// TwinCAT 3 PLC project PLC1
// ProgramVersion: 3.1.4024.0
// libraries:
//   Tc2_HVAC, * (Beckhoff Automation GmbH)
//   Tc2_Math, * (Beckhoff Automation GmbH)
//   Tc2_MC2, * (Beckhoff Automation GmbH)
//   Tc2_Standard, * (Beckhoff Automation GmbH)
//   Tc2_System, * (Beckhoff Automation GmbH)
//   Tc2_TcpIp, * (Beckhoff Automation GmbH)
//   Tc2_Utilities, * (Beckhoff Automation GmbH)
//   Tc3_Module, * (Beckhoff Automation GmbH)
// project tree:
//   DUTs/ E_6Axis_Command.TcDUT, E_6Axis_Motion.TcDUT, E_ConnectionSteps.TcDUT, getPosition.TcDUT, Motion_Command_Input.TcDUT, ST_6Axis_State.TcDUT
//   GVLs/ AutoMotionData.TcGVL, GVL.TcGVL
//   / PlcTask.TcTTO
//   POUs/Airbus_TCP/ Deserialize.TcPOU, FB_TCPClient.TcPOU, Serialize.TcPOU
//   POUs/ Buffer.TcPOU, MC_Linear.TcPOU, Kinematics.TcPOU, MAIN.TcPOU, Controller.TcPOU, MathFunc.TcPOU
// real-time tasks:
//   TASK PlcTask: cycle T#2ms, priority 20, ADS port 350
// motion (NC):
//   TASK NC-Task 1 SAF: cycle T#2ms, priority 4, ADS port 501
//   TASK NC-Task 1 SVB: cycle T#10ms, priority 8, ADS port 511
//   AXIS Axis 1 (id 1)
//     Dynamic: AccelerationMaximum=1500, DecelerationMaximum=1500
//     Velo: RefSearch=1, RefSync=1, SlowManual=1, FastManual=3, Maximum=45
//     OtherSettings: AllowMotionCmdToSlave=true
//     encoder EncType=1
//       EncPara: ScaleFactorNumerator=360, ScaleFactorDenominator=104857600, EncMode=3
//         SoftEndMinControl: Enable=true, Range=-180
//         SoftEndMaxControl: Enable=true, Range=180
//     drive DrvType=5
//       Analog: VeloReferenz=50, TorqueSetpointScale=10, ScaleFactorActTorque=0.1
//       TimeComp: TaskDelayCycles=1
//     controller CtrType=1
//       CtrPara: PriorControlFactor=1
//         Observer: BandWidth=20
//   AXIS Axis 2 (id 2)
//     Velo: RefSearch=1, RefSync=1, SlowManual=1, FastManual=3, Maximum=30
//     OtherSettings: AllowMotionCmdToSlave=true
//     encoder EncType=1
//       EncPara: ScaleFactorNumerator=360, ScaleFactorDenominator=104857600, Offset=-0.1609, EncMode=3
//         SoftEndMinControl: Enable=true, Range=-57
//         SoftEndMaxControl: Enable=true, Range=120
//     drive DrvType=5
//       Analog: VeloReferenz=40, TorqueSetpointScale=10, ScaleFactorActTorque=0.1
//       TimeComp: TaskDelayCycles=1
//     controller CtrType=1
//       CtrPara: PriorControlFactor=1
//         Observer: BandWidth=20
//   AXIS Axis 3 (id 3)
//     Velo: RefSearch=1, RefSync=1, SlowManual=1, FastManual=3, Maximum=30
//     OtherSettings: AllowMotionCmdToSlave=true
//     encoder EncType=1
//       EncPara: ScaleFactorNumerator=360, ScaleFactorDenominator=83886080, Offset=2.384, EncMode=3
//         SoftEndMinControl: Enable=true, Range=-125
//         SoftEndMaxControl: Enable=true, Range=55
//     drive DrvType=5
//       Analog: VeloReferenz=40, TorqueSetpointScale=10, ScaleFactorActTorque=0.1
//       TimeComp: TaskDelayCycles=1
//     controller CtrType=1
//       CtrPara: PriorControlFactor=1
//         Observer: BandWidth=20
//   AXIS Axis 4 (id 4)
//     Velo: RefSearch=1, RefSync=1, SlowManual=1, FastManual=3, Maximum=80
//     OtherSettings: AllowMotionCmdToSlave=true
//     encoder EncType=1
//       EncPara: ScaleFactorNumerator=360, ScaleFactorDenominator=83886080, Offset=0.2524, EncMode=3
//         SoftEndMinControl: Enable=true, Range=-180
//         SoftEndMaxControl: Enable=true, Range=180
//     drive DrvType=5
//       Analog: VeloReferenz=100, TorqueSetpointScale=10, ScaleFactorActTorque=0.1
//       TimeComp: TaskDelayCycles=1
//     controller CtrType=1
//       CtrPara: PriorControlFactor=1
//         Observer: BandWidth=20
//   AXIS Axis 5 (id 5)
//     Velo: RefSearch=1, RefSync=1, SlowManual=1, FastManual=3, Maximum=50
//     OtherSettings: AllowMotionCmdToSlave=true
//     encoder EncType=1
//       EncPara: ScaleFactorNumerator=360, ScaleFactorDenominator=64225280, Offset=0.9798, EncMode=3
//         SoftEndMinControl: Enable=true, Range=-95
//         SoftEndMaxControl: Enable=true, Range=95
//     drive DrvType=5
//       Analog: VeloReferenz=60, TorqueSetpointScale=10, ScaleFactorActTorque=0.1
//       TimeComp: TaskDelayCycles=1
//     controller CtrType=1
//       CtrPara: PriorControlFactor=1
//         Observer: BandWidth=20
//   AXIS Axis 6 (id 6)
//     Velo: RefSearch=1, RefSync=1, SlowManual=1, FastManual=3, Maximum=30000
//     OtherSettings: AllowMotionCmdToSlave=true
//     encoder EncType=1
//       EncPara: ScaleFactorNumerator=360, ScaleFactorDenominator=52428800, Offset=-113, EncMode=3
//         SoftEndMinControl: Enable=true, Range=-180
//         SoftEndMaxControl: Enable=true, Range=180
//     drive DrvType=5
//       Analog: VeloReferenz=30000, TorqueSetpointScale=10, ScaleFactorActTorque=0.1
//       TimeComp: TaskDelayCycles=1
//     controller CtrType=1
//       CtrPara: PriorControlFactor=1
//         Observer: BandWidth=20
// I/O:
//   DEVICE Device 2 (EtherCAT) (disabled), AmsNetId 169.254.73.89.3.1
//     Term 1 (R1-EC5500) [R1-EC5500 EtherCAT to E-BUS adapter Module]
//       Term 2 (R1-EC6022) [R1-EC6022 16-ch Sink/Source Type Digital Input Module with 2ms Filter Function]
//       Term 3 (R1-EC7062) [R1-EC7062 16-ch 24VDC/0.5A/Sink Type Digital Output Module]
//       Term 4 (R1-EC8124D0) [R1-EC8124D0 4-ch 16-bit Single-ended/10kHz/Voltage or Current Mode A/D Control Module]
//       Term 11 (EL9011) [EL9011 End Terminal]
//     Drive 5 (SGD7S-xxxxA0x CoE Drive) [SGD7S-xxxxA0x EtherCAT(CoE) SERVOPACK Rev6.01]
//     Drive 6 (SGD7S-xxxxA0x CoE Drive) [SGD7S-xxxxA0x EtherCAT(CoE) SERVOPACK Rev6.01]
//     Drive 7 (SGD7S-xxxxA0x CoE Drive) [SGD7S-xxxxA0x EtherCAT(CoE) SERVOPACK Rev8.19]
//     Drive 8 (SGD7S-xxxxA0x CoE Drive) [SGD7S-xxxxA0x EtherCAT(CoE) SERVOPACK Rev6.01]
//     Drive 9 (SGD7S-xxxxA0x CoE Drive) [SGD7S-xxxxA0x EtherCAT(CoE) SERVOPACK Rev6.01]
//     Drive 10 (SGD7S-xxxxA0x CoE Drive) [SGD7S-xxxxA0x EtherCAT(CoE) SERVOPACK Rev6.01]
// variable links:
//   PLC1/PLC1 Instance <-> NC-Task 1 SAF/Axes/Axis 1
//     PlcTask Inputs/MAIN.SixAxis.Axis[1].NcToPlc <-> Outputs/ToPlc
//     PlcTask Outputs/MAIN.SixAxis.Axis[1].PlcToNc <-> Inputs/FromPlc
//   PLC1/PLC1 Instance <-> NC-Task 1 SAF/Axes/Axis 2
//     PlcTask Inputs/MAIN.SixAxis.Axis[2].NcToPlc <-> Outputs/ToPlc
//     PlcTask Outputs/MAIN.SixAxis.Axis[2].PlcToNc <-> Inputs/FromPlc
//   PLC1/PLC1 Instance <-> NC-Task 1 SAF/Axes/Axis 3
//     PlcTask Inputs/MAIN.SixAxis.Axis[3].NcToPlc <-> Outputs/ToPlc
//     PlcTask Outputs/MAIN.SixAxis.Axis[3].PlcToNc <-> Inputs/FromPlc
//   PLC1/PLC1 Instance <-> NC-Task 1 SAF/Axes/Axis 4
//     PlcTask Inputs/MAIN.SixAxis.Axis[4].NcToPlc <-> Outputs/ToPlc
//     PlcTask Outputs/MAIN.SixAxis.Axis[4].PlcToNc <-> Inputs/FromPlc
//   PLC1/PLC1 Instance <-> NC-Task 1 SAF/Axes/Axis 5
//     PlcTask Inputs/MAIN.SixAxis.Axis[5].NcToPlc <-> Outputs/ToPlc
//     PlcTask Outputs/MAIN.SixAxis.Axis[5].PlcToNc <-> Inputs/FromPlc
//   PLC1/PLC1 Instance <-> NC-Task 1 SAF/Axes/Axis 6
//     PlcTask Inputs/MAIN.SixAxis.Axis[6].NcToPlc <-> Outputs/ToPlc
//     PlcTask Outputs/MAIN.SixAxis.Axis[6].PlcToNc <-> Inputs/FromPlc

CONFIGURATION PLC1
    RESOURCE PLC ON TwinCAT3
        TASK PlcTask(INTERVAL := T#2ms, PRIORITY := 20);
        PROGRAM MAIN WITH PlcTask : MAIN;
    END_RESOURCE
END_CONFIGURATION

// ---- DUTs/E_6Axis_Command.TcDUT
{attribute 'qualified_only'}
{attribute 'strict'}
TYPE E_6Axis_Command :
(
	NO_COMMAND,
	POWER_ON,
	STOP,
	HALT,
	RESET,
	HOMING,
	// Command For Testing
	M_PTP,
	M_DIRE_X,
	M_DIRE_Y,
	M_DIRE_XY,
	M_DIRE_Z,
	M_LINEAR,
	M_CURVE,
	CONSTRUCT, //To build Jenga
	LOOKING,   //To observe Jenga
	TOUCHING,  //To detech Jenga status
	TAKING     //To clamping Jenga
) := NO_COMMAND;
END_TYPE

// ---- DUTs/E_6Axis_Motion.TcDUT
TYPE E_6Axis_Motion :
(
	PTP,
	LINEAR,
	CURVE
);
END_TYPE

// ---- DUTs/E_ConnectionSteps.TcDUT
TYPE E_ConnectionSteps :
(
	eCONNECTION_STATE_IDLE,
	eCONNECTION_STATE_CONNECT_START,
	eCONNECTION_STATE_CONNECT_WAIT,
	eCONNECTION_STATE_DATAEXCHANGE,
	eCONNECTION_STATE_CLOSE_START,
	eCONNECTION_STATE_CLOSE_WAIT,
	eCONNECTION_STATE_ERROR
);
END_TYPE

// ---- DUTs/getPosition.TcDUT
TYPE getPosition :
STRUCT
	a : BYTE;
	b : DINT;
	c : ARRAY[1..6] OF LREAL;
END_STRUCT
END_TYPE

// ---- DUTs/Motion_Command_Input.TcDUT
TYPE Motion_Command_Input :
STRUCT
	mode : E_6Axis_Motion;
	precise : BOOL; // 專門給Homing指令使用
	StartPOS : ARRAY [1..6] OF LREAL;
	FinalPOS : ARRAY [1..6] OF LREAL;
	
END_STRUCT
END_TYPE

// ---- DUTs/ST_6Axis_State.TcDUT
TYPE ST_6Axis_State :
STRUCT
	ready : BOOL;
	busy : BOOL;
	error : BOOL;
	powerOn : BOOL;
	stop : BOOL;
	moving : BOOL;
END_STRUCT
END_TYPE

// ---- GVLs/AutoMotionData.TcGVL
{attribute 'qualified_only'}
VAR_GLOBAL
	POStore : ARRAY [1..2] OF ARRAY [0..100] OF ARRAY [1..6] OF LREAL := [
		[[559, 13, 400, 0, 90, -45]],
		[[561, -43, 400, 0, 90, -135]]];
	MovableBlocks : ARRAY [1..100] OF ARRAY [1..6] OF LREAL; 
	
	CAMStore : ARRAY [1..3] OF ARRAY [0..100] OF ARRAY [1..6] OF LREAL := [
	    [[559, 13, 400, 0, 135, -45]],
		[[561, -43, 400, 0, 135, -135]]]; //姿態要改 
	Heightstore : ARRAY [1..1] OF LREAL ;
END_VAR

// ---- GVLs/GVL.TcGVL
VAR_GLOBAL
	// Software
	isHalt : BOOL;
	InitalPOS : ARRAY [1..6] OF LREAL;

	//Hardward
	input_ana AT %I* : ARRAY[1..8] OF INT;
	output_dig AT %Q* : ARRAY[1..16] OF BOOL;
	input_dig AT %I* : ARRAY[1..16] OF BOOL;
	
	// Extend DATA feat. ADS
	ExtData AT %I* : DINT;
	
	// Extend DATA feat. TCP
	aaa : STRING;
	
END_VAR	
	
VAR_GLOBAL CONSTANT
	// Axes Number
	AXIS_MIN_IDX : USINT := 1;
	AXIS_MAX_IDX : USINT := 6;

	// ADS Setting
	
	// TCP Setting
	PLCPRJ_BUFFER_SIZE						: UDINT := 1000;
	PLCPRJ_SEND_CYCLE_TIME					: TIME := T#1S;
	PLCPRJ_RECEIVE_POLLING_TIME		 		: TIME := T#100MS;
	PLCPRJ_RECEIVE_TIMEOUT					: TIME := T#50S;
	(* Some project specific error codes *)
	PLCPRJ_ERROR_RECEIVE_TIMEOUT			: UDINT := 16#8101;(* Receive timeout error *)
	PLCPRJ_ERROR_SENDFIFO_OVERFLOW			: UDINT := 16#8102;(* Send fifo overflow *)
	PLCPRJ_ERROR_RECFIFO_OVERFLOW			: UDINT := 16#8103;(* Receive fifo overflow *)

END_VAR

// ---- POUs/MAIN.TcPOU
PROGRAM MAIN  
// vision 4.4 *+: TCP, 斜直線移動

VAR
	SixAxis : Controller;
	readA : REAL;
	
	bInit: BOOL := TRUE;
	fbSocketCloseAll: FB_SocketCloseAll; 
	serialize : Serialize;
	deserialize : Deserialize;
	bSocketCloseError: BOOL;
	nSocketCloseError: UDINT;
	
	TCP_Client1     				: FB_TCPClient;
		sClient1SendData			: ARRAY[0..1023] OF BYTE;
		sServer1Host				: T_IPv4Addr;
		nServer1Port				: UDINT;
		bStartClient1Communication	: BOOL 			    := TRUE;
		tClient1CycleTime			: TIME 				:= T#0.5S;
		bClient1SendTrigger			: BOOL;
		bClient1Connected			: BOOL;
		sClient1ReceivedData		: ARRAY[0..1023] OF BYTE;
		bClient1Busy				: BOOL;
		bClientError1				: BOOL;
		nClient1ErrorID1			: UDINT;
		// 新增內容
		rx                          : BYTE;
		mode                        : DINT;
		position                    : ARRAY[1..6] OF LREAL;  // xyzrpy
		tx                          : BYTE;
		fullTime                    : LREAL;
		coeffCopy                   : ARRAY[1..6, 1..6] OF LREAL;
	bAutogenerateData				: BOOL 				:= TRUE;
	fbTimer1						: TON;
	simTime                         : DINT;
	simCoeff                        : ARRAY[1..6] OF LREAL;
	nCnt							: UDINT;	
	
END_VAR

















//	L1 : ARRAY [1..6,1..6] OF LREAL;
//	L2 : ARRAY [1..6,1..6] OF LREAL;
//	L6 : ARRAY [1..6,1..6] OF LREAL;
//	L3,L5 : ARRAY [1..2] OF LREAL;
//	L4 : ARRAY [1..2] OF LREAL := [1, 2];
	
//	i: INT;
//	j: INT;
//	k : Lreal;

SixAxis();
//readA := (INT_TO_REAL(GVL.input_ana[1]) / 32767) * 10;

// Transmission Program
(* On PLC reset or program download close all created/opened sockets/connections *)
// Init Step to close all sockets after login PLC with  downlaod
sServer1Host := '192.168.1.47';
nServer1Port := 200;

IF bInit THEN 			
	fbSocketCloseAll(
		sSrvNetId:= '', 
		bExecute:= TRUE, 
		tTimeout:= T#3S, 
		bBusy=> , 
		bError=> bSocketCloseError, 
		nErrId=> nSocketCloseError);
	IF NOT (fbSocketCloseAll.bBusy OR fbSocketCloseAll.bError) THEN
		bInit := FALSE;
		fbSocketCloseAll(bExecute:= FALSE);
	END_IF
ELSE
	TCP_Client1(
		nRemotePort:= nServer1Port, 								// Server port
		sRemoteHost:= sServer1Host, 								// Server IP (empty for local communication)
		bStartCommunication:= bStartClient1Communication, 			// Start communication, when FALSE, connection is closed
		sSendData:= sClient1SendData, 								// Data that are sent to the server
		tCycleTimeSend:= (*tClient1CycleTime*), 					// TimeInterval for cyclic sending
		bSendTrigger:= ,											// Trigger to send one telegramm manually 
		bConnected => bClient1Connected,							// Switches to TRUE when Client is connected to a server
		sReceivedData=> sClient1ReceivedData,						// Data that are received
		bBusy=> bClient1Busy, 
		bError=> bClientError1, 
		nErrorID=> nClient1ErrorID1, ); 
	deserialize(
		Recvbuffer := sClient1ReceivedData,
		a => rx,
		b => mode,
		c => position);
	
	IF bAutogenerateData AND bClient1Connected THEN
		fbTimer1(IN:= NOT fbTimer1.Q, PT:= tClient1CycleTime, Q=> , ET=> );
		IF fbTimer1.Q  THEN
			IF rx = 84 THEN
				SixAxis.SetMotion(
					mode, SixAxis.HomePoint, position, TRUE, FALSE,
					runTime => fullTime,
					coeffCopy => coeffCopy);
				tx := 67;
				serialize(
					a := tx,
					b := fullTime,
					c := coeffCopy,
					sendbuffer => sClient1SendData);
			
			END_IF
			TCP_Client1.bSendTrigger := TRUE;
			nCnt := nCnt + 1;
		ELSE
			TCP_Client1.bSendTrigger := FALSE;
		END_IF
	END_IF 
END_IF
























// 測試KM
//k := 1.235415445;
//k := LREAL_TO_DINT(k*EXPT(10,2) )/EXPT(10,2);
//FOR i := 1 TO 6 DO
//	FOR j := 1 TO 6 DO
//		IF i <= j THEN
//			L1[i, j] := j;
//		ELSE
//			L1[i, j] := i;
//		END_IF
//	END_FOR
//END_FOR

//FOR i := 1 TO 6 DO
//	FOR j := 1 TO 6 DO
//		IF i <= j THEN
//			L2[i, j] := i*j;
//		ELSE
//			L2[i, j] := i*i;
//		END_IF
//	END_FOR
//END_FOR

////MF.GaussianElimination(base_mat := L1, extend_mat := L2, temp_mat := L6, 6);

END_PROGRAM

// ---- POUs/Controller.TcPOU
FUNCTION_BLOCK Controller

VAR_OUTPUT
	
END_VAR

VAR	
	// 輸入指令，顯示狀態、位置、角度
	command : E_6Axis_Command;	
	state : ST_6Axis_State;
	constructState : UINT;
	touchingState : UINT;
	takeState : UINT;
	JointDegNow : ARRAY [AXIS_MIN_IDX..AXIS_MAX_IDX] OF LREAL;
	PositionNow : ARRAY [AXIS_MIN_IDX..AXIS_MAX_IDX] OF LREAL;
	hasFromCAM : BOOL;
	//StartPosition_Now : ARRAY [AXIS_MIN_IDX..AXIS_MAX_IDX] OF LREAL; // for linear move used
	
	// 開發者使用
	HomePoint : ARRAY [AXIS_MIN_IDX..AXIS_MAX_IDX] OF LREAL := [565, 0, 834, 0, 0, 0];
	HomeJoint : ARRAY [AXIS_MIN_IDX..AXIS_MAX_IDX] OF LREAL := [0, 0, 0, 0, 0, 0]; // for joints space	

	//BufferMot : Motion_Command_Input; // 
	InitalPOS : ARRAY [AXIS_MIN_IDX..AXIS_MAX_IDX] OF LREAL := InitalPOS;
	ActExecute : BOOL := FALSE;
	ExecutePMD : BOOL := FALSE;
	ExecuteCAL : BOOL := FALSE; // 執行一次性計算
 	DIR : LREAL := 0; // XYZ_Direcation XYZ軸方向 = {1:x, 2:y, 3:z, 4:xy, 5:-(xy)}
	PMD : LREAL := 0; // Path_Motion_Displace 路徑移動距離
	TouchDetection : BOOL;
	ZeroArray : ARRAY [AXIS_MIN_IDX..AXIS_MAX_IDX] OF LREAL := [0, 0, 0, 0, 0, 0]; 
	TargetPOS : ARRAY [AXIS_MIN_IDX..AXIS_MAX_IDX] OF LREAL := [650, -150, 500, -42, 0, 45];
	POS_STORAGE : Buffer;

	// 索引
	idx : USINT(AXIS_MIN_IDX..AXIS_MAX_IDX);
	movableBlock_idx : INT;
	i, j : USINT(AXIS_MIN_IDX..AXIS_MAX_IDX);
	z : INT;
	n : ARRAY [1..6] OF LREAL := AutoMotionData.CAMStore[1][0] ;
	usingMotion : INT;
	row, col : INT;
	//ok
	//p : ARRAY [1..2] OF LREAL := AutoMotionData.CAMStore;
	//L : ARRAY [AXIS_MIN_IDX..AXIS_MAX_IDX] OF LREAL ;
	h : INT;
	

	// 基本需要的函式
	Axis : ARRAY[AXIS_MIN_IDX..AXIS_MAX_IDX] OF AXIS_REF;
	Power : ARRAY [AXIS_MIN_IDX..AXIS_MAX_IDX] OF MC_Power;
	Stop : ARRAY [AXIS_MIN_IDX..AXIS_MAX_IDX] OF MC_Stop; //delete
	Halt : ARRAY [AXIS_MIN_IDX..AXIS_MAX_IDX] OF MC_Halt; 
	Reset : ARRAY [AXIS_MIN_IDX..AXIS_MAX_IDX] OF MC_Reset;
	
	// 自訂義函式
	KM : Kinematics;
	MF : MathFunc;
	
	// 移動用函式
	AbsMove : ARRAY [AXIS_MIN_IDX..AXIS_MAX_IDX] OF MC_MoveAbsolute;
	ExtSwitchEn : ARRAY [AXIS_MIN_IDX..AXIS_MAX_IDX] OF MC_ExtSetPointGenEnable;
	ExtSwitchDis : ARRAY [AXIS_MIN_IDX..AXIS_MAX_IDX] OF MC_ExtSetPointGenDisable;
	LinearMove : MC_Linear; 

	// For Curve                         A1  A2  A3  A4  A5  A6
	StartVEL : ARRAY [1..6] OF LREAL := [  0,  0,  0,  0,  0,  0];
	StartACC : ARRAY [1..6] OF LREAL := [  0,  0,  0,  0,  0,  0];
	FinalVEL : ARRAY [1..6] OF LREAL := [  0,  0,  0,  0,  0,  0];
	FinalACC : ARRAY [1..6] OF LREAL := [  0,  0,  0,  0,  0,  0];

	E_Command: INT;
	No_Command: INT;
	PT: TIME;
END_VAR

readAxis();
SetStartPosition();

CASE command OF
	E_6Axis_Command.NO_COMMAND:
		FOR idx := AXIS_MIN_IDX TO AXIS_MAX_IDX DO
			AbsMove[idx].Execute := FALSE;
		END_FOR
		isHalt := FALSE;
		ExecutePMD := FALSE;
		constructState := 0;
		ActExecute := FALSE;
		
	E_6Axis_Command.POWER_ON:
		FOR idx := AXIS_MIN_IDX TO AXIS_MAX_IDX DO
			Power[idx].Enable := TRUE;
		END_FOR
		IF state.powerOn THEN
			command := E_6Axis_Command.HOMING;
		END_IF
	
	E_6Axis_Command.HALT:
		FOR idx := AXIS_MIN_IDX TO AXIS_MAX_IDX DO
			Halt[idx].Execute := TRUE;
		END_FOR
		IF NOT state.moving THEN
			FOR idx := AXIS_MIN_IDX TO AXIS_MAX_IDX DO
				Halt[idx].Execute := FALSE;
			END_FOR
		END_IF
		command := E_6axis_Command.NO_COMMAND;
	
	E_6Axis_Command.RESET:
		FOR idx := AXIS_MIN_IDX TO AXIS_MAX_IDX DO
			Reset[idx].Execute := TRUE;
			IF Reset[idx].Done THEN
				Reset[idx].Execute := FALSE;
			END_IF
		END_FOR
		command := E_6axis_Command.NO_COMMAND;

	// SetMotion(路徑模式，起點，終點，FALSE);		
	E_6Axis_Command.HOMING:
		ActExecute := TRUE;
		SetMotion(0, InitalPOS, HomeJoint, FALSE, TRUE);
		IF NOT ActExecute THEN
			command := E_6axis_Command.NO_COMMAND;
		END_IF

	E_6Axis_Command.M_PTP:
		ActExecute := TRUE;
		SetMotion(0, InitalPOS, TargetPOS, FALSE, FALSE);
		IF NOT ActExecute THEN
			command := E_6axis_Command.NO_COMMAND;
		END_IF
		
	E_6Axis_Command.M_DIRE_X:
		IF NOT ExecutePMD THEN
			MF.VectorMotionPOS(POS := TargetPOS, DIR, PMD);
			ExecutePMD := TRUE;
		END_IF
		ActExecute := TRUE;
		SetMotion(1, InitalPOS, TargetPOS, FALSE, FALSE);
		IF NOT ActExecute THEN
			command := E_6axis_Command.NO_COMMAND;
		END_IF
		
	E_6Axis_Command.M_DIRE_Y:
		IF NOT ExecutePMD THEN
			MF.VectorMotionPOS(POS := TargetPOS, DIR, PMD);
			ExecutePMD := TRUE;
		END_IF
		ActExecute := TRUE;
		SetMotion(1, InitalPOS, TargetPOS, FALSE, FALSE);
		IF NOT ActExecute THEN
			command := E_6axis_Command.NO_COMMAND;
		END_IF
	
	E_6Axis_Command.M_DIRE_XY:
		IF NOT ExecutePMD THEN
			MF.VectorMotionPOS(POS := TargetPOS, DIR, PMD);
			ExecutePMD := TRUE;
		END_IF
		ActExecute := TRUE;
		SetMotion(1, InitalPOS, TargetPOS, FALSE, FALSE);
		IF NOT ActExecute THEN
			command := E_6axis_Command.NO_COMMAND;
		END_IF
		
	E_6Axis_Command.M_DIRE_Z:
		IF NOT ExecutePMD THEN
			MF.VectorMotionPOS(POS := TargetPOS, DIR, PMD);
			ExecutePMD := TRUE;
		END_IF
		ActExecute := TRUE;
		SetMotion(1, InitalPOS, TargetPOS, FALSE, FALSE);
		IF NOT ActExecute THEN
			command := E_6axis_Command.NO_COMMAND;
		END_IF
		
	E_6Axis_Command.M_LINEAR:
		ActExecute := TRUE;
		SetMotion(1, InitalPOS, TargetPOS, FALSE, FALSE);
		IF NOT ActExecute THEN
			command := E_6axis_Command.NO_COMMAND;
		END_IF
		
	E_6Axis_Command.M_CURVE:
		ActExecute := TRUE;
		SetMotion(2, InitalPOS, TargetPOS, FALSE, FALSE);
		IF NOT ActExecute THEN
			command := E_6axis_Command.NO_COMMAND;
		END_IF
		
	E_6Axis_Command.TOUCHING://判斷式
		IF NOT ActExecute THEN
			CASE touchingState OF
				0: //要再加一個判斷式判斷是哪一個位置
					//z := z + 1;            // 疊疊樂右面與左面
					usingMotion := 2;
					
					IF z = 1 THEN
						TargetPOS[1]:= n[1];
						TargetPOS[2]:= n[2];
						TargetPOS[3]:= 500;
						TargetPOS[4]:= 0;
						TargetPOS[5]:= 90;
						TargetPOS[6]:= -45;
					ELSIF z = 2 THEN
						TargetPOS[1]:= n[1];
						TargetPOS[2]:= n[2];
						TargetPOS[3]:= 500;
						TargetPOS[4]:= 0;
						TargetPOS[5]:= 90;
						TargetPOS[6]:= -135;
					END_IF
					      // 移動模式
					//TargetPOS := AutoMotionData.CAMStore[n][z];  // n=0
					//n := n + 1;
					touchingState := touchingState + 1;
				1:
					usingMotion := 1;
					IF z = 1 THEN
						MF.VectorMotionPOS(POS := TargetPOS, 5, -25);
					ELSIF z = 2 THEN
						MF.VectorMotionPOS(POS := TargetPOS, 4, 25);
					END_IF
					//AutoMotionData.POStore[z][n] := TargetPOS;
					//n := n + 1;
					touchingState := touchingState + 1;
				2: 
					usingMotion := 1;
					IF z = 1 THEN
						MF.VectorMotionPOS(POS := TargetPOS, 3, -(500-n[3]));
					ELSIF z = 2 THEN
						MF.VectorMotionPOS(POS := TargetPOS, 3, -(500-n[3]));
					END_IF
					touchingState := touchingState + 1;
				3:
					PT := T#1S;
					input_dig[1] := TRUE;
					PT := T#1S;
					//加計時器
					input_dig[1] := FALSE;
				4:
					usingMotion := 1;
					IF z = 1 THEN
						MF.VectorMotionPOS(POS := TargetPOS, 3, (500-n[3]));
					ELSIF z = 2 THEN
						MF.VectorMotionPOS(POS := TargetPOS, 3, (500-n[3]));
					END_IF
					touchingState := touchingState + 1;
				
				5:
					command := E_6axis_Command.HOMING;
					touchingState := touchingState + 1;
				6:
					command := E_6axis_Command.TAKING;
			END_CASE			
		END_IF
	SetMotion(usingMotion, InitalPOS, TargetPOS, FALSE, FALSE);
	
	E_6Axis_Command.TAKING:
		IF NOT ActExecute THEN
			CASE takeState OF
				0:
					usingMotion := 1;
					input_dig[2] := FALSE;
					
					IF z = 1 THEN
						MF.VectorMotionPOS(POS := TargetPOS, 5, (n[1]+100));
						MF.VectorMotionPOS(POS := TargetPOS, 5, (n[2]+100));
						TargetPOS[3] := 500;
						TargetPOS[4] := 0;
						TargetPOS[5] := -90;
						TargetPOS[6] := 45;
					ELSIF z = 2 THEN
						MF.VectorMotionPOS(POS := TargetPOS, 4, (n[1]-100));
						MF.VectorMotionPOS(POS := TargetPOS, 4, (n[2]-100));
						TargetPOS[3] := 500;
						TargetPOS[4] := 0;
						TargetPOS[5] := -90;
						TargetPOS[6] := -135;
						
					END_IF
					touchingState := touchingState + 1;	
				1:
					usingMotion := 1;
					IF z = 1 THEN
						MF.VectorMotionPOS(POS := TargetPOS, 3, -(500-n[3]));
					ELSIF z = 2 THEN
						MF.VectorMotionPOS(POS := TargetPOS, 3, -(500-n[3]));
					END_IF
					//AutoMotionData.POStore[z][n] := hasFromCAM;
					//n := n + 1;
					touchingState := touchingState + 1;
				2:
					usingMotion := 1; 
					input_dig[2]:= TRUE ;
					PT := T#1S;
					touchingState := touchingState + 1;
				3:
					usingMotion := 1; 
					IF z = 1 THEN
						MF.VectorMotionPOS(POS := TargetPOS, 5, 30);
					ELSIF z = 2 THEN
						MF.VectorMotionPOS(POS := TargetPOS, 4, -30);
					END_IF
					touchingState := touchingState + 1;
				4:
					usingMotion := 1;
					
					MF.VectorMotionPOS(POS := TargetPOS, 3, (AutoMotionData.Heightstore[1]-n[3]+2));
					touchingState := touchingState + 1;
				5:
				   IF z = 1 THEN
						MF.VectorMotionPOS(POS := TargetPOS, 5, -60);
					ELSIF z = 2 THEN
						MF.VectorMotionPOS(POS := TargetPOS, 4, 60);
					END_IF
					PT := T#1S;
					input_dig[2]:= FALSE ;
					touchingState := touchingState + 1;
				6:
					command := E_6axis_Command.HOMING;
					
			END_CASE
		END_IF
		SetMotion(usingMotion, InitalPOS, TargetPOS, FALSE, FALSE);
		ActExecute := TRUE;
				
				
//	E_6Axis_Command.LOOKING:
//		SetMotion(0, InitalPOS, TargetPOS, FALSE);

END_CASE

Decider();
Update_AbsMove_Motion();
Update_Custom_Motion();
ActPower();
ActReset();
ActStop();

//	E_6Axis_Command.CONSTRUCT:
//		IF NOT ActExecute THEN
//			CASE constructState OF
//				0:
//					z := z + 1;            // 疊疊樂右面與左面
//					usingMotion := 2;      // 移動模式
//					TargetPOS := AutoMotionData.POStore[z][n];  // n=0
//					n := n + 1;
//					constructState := constructState + 1;
//				1:
//					usingMotion := 1;
//					IF z = 1 THEN
//						MF.VectorMotionPOS(POS := TargetPOS, 4, 90);
//					ELSIF z = 2 THEN
//						MF.VectorMotionPOS(POS := TargetPOS, 5, 90);
//					END_IF
//					AutoMotionData.POStore[z][n] := TargetPOS;
//					n := n + 1;
//					constructState := constructState + 1;
//				2:
//					usingMotion := 1;
//					IF z = 1 THEN
//						MF.VectorMotionPOS(POS := TargetPOS, 3, -95);
//					ELSIF z = 2 THEN
//						MF.VectorMotionPOS(POS := TargetPOS, 3, -110);
//					END_IF					
//					AutoMotionData.POStore[z][n] := TargetPOS;
//					n := n + 1;
//					constructState := constructState + 1;
//				3:
//					usingMotion := 1;
//					TouchDetection := TRUE;
//					ExecuteCAL := FALSE;
//					IF z = 1 THEN
//						MF.VectorMotionPOS(POS := TargetPOS, 4, -40);
//					ELSIF z = 2 THEN
//						MF.VectorMotionPOS(POS := TargetPOS, 5, -40);
//					END_IF	
//					AutoMotionData.POStore[z][n] := TargetPOS;
//					n := n + 1;
//					movableBlock_idx := movableBlock_idx + 1;
//					constructState := constructState + 1;
//				4:
//					usingMotion := 1;
//					TouchDetection := FALSE;
//					row := row + 1;
//					IF z = 1 THEN
//						MF.VectorMotionPOS(POS := TargetPOS, 4, 40);
//					ELSIF z = 2 THEN
//						MF.VectorMotionPOS(POS := TargetPOS, 5, 40);
//					END_IF	
//					AutoMotionData.POStore[z][n] := TargetPOS;
//					n := n + 1; 
//					constructState := constructState + 1;
//					IF row = 3 THEN
//						row := 0;
//						constructState := 6;
//						col := col + 1;
//						IF col = 4 THEN
//							constructState := 8;
//						END_IF
//					END_IF
//				5:
//					usingMotion := 1;
//					IF z = 1 THEN
//						MF.VectorMotionPOS(POS := TargetPOS, 5, -25);
//					ELSIF z = 2 THEN
//						MF.VectorMotionPOS(POS := TargetPOS, 4, -25);
//					END_IF	
//					AutoMotionData.POStore[z][n] := TargetPOS;
//					n := n + 1;
//					constructState := 3;
//				6:
//					usingMotion := 1;
//					MF.VectorMotionPOS(POS := TargetPOS, 3, -30);
//					AutoMotionData.POStore[z][n] := TargetPOS;
//					n := n + 1;
//					constructState := constructState + 1;
//				7:
//					usingMotion := 1;
//					IF z = 1 THEN
//						MF.VectorMotionPOS(POS := TargetPOS, 5, 50);
//					ELSIF z = 2 THEN
//						MF.VectorMotionPOS(POS := TargetPOS, 4, 50);
//					END_IF	
//					AutoMotionData.POStore[z][n] := TargetPOS;
//					n := n + 1;
//					constructState := 3;
//				8:
//					usingMotion := 2;
//					TargetPOS := AutoMotionData.POStore[z][1];
//					constructState := 9;
//				9:
//					usingMotion := 2;
//					TargetPOS := HomePoint;
//					n := 0;
//					row := 0;
//					col := 0;
//					constructState := 0;
//					IF z = 2 THEN
//						constructState := 10;
//					END_IF
//				10:
//					command := E_6axis_Command.HOMING;
//					constructState := 11;
//			END_CASE
//		END_IF
//		ActExecute := TRUE;
//		IF TouchDetection THEN
//			IF input_dig[1] THEN
//				IF NOT ExecuteCAL THEN
//					AutoMotionData.MovableBlocks[movableBlock_idx] := ZeroArray;
//					movableBlock_idx := movableBlock_idx - 1;
//					ExecuteCAL := TRUE;
//				END_IF
//			ELSE
//				// 減2是為了擷取上一個座標
//				AutoMotionData.MovableBlocks[movableBlock_idx] := AutoMotionData.POStore[z][n-2];
//			END_IF
//		END_IF

//		IF NOT (constructState = 11) THEN
//			SetMotion(usingMotion, InitalPOS, TargetPOS, FALSE, FALSE);
//		ELSE
//			z := 0;
//		END_IF

ACTION ActHalt:
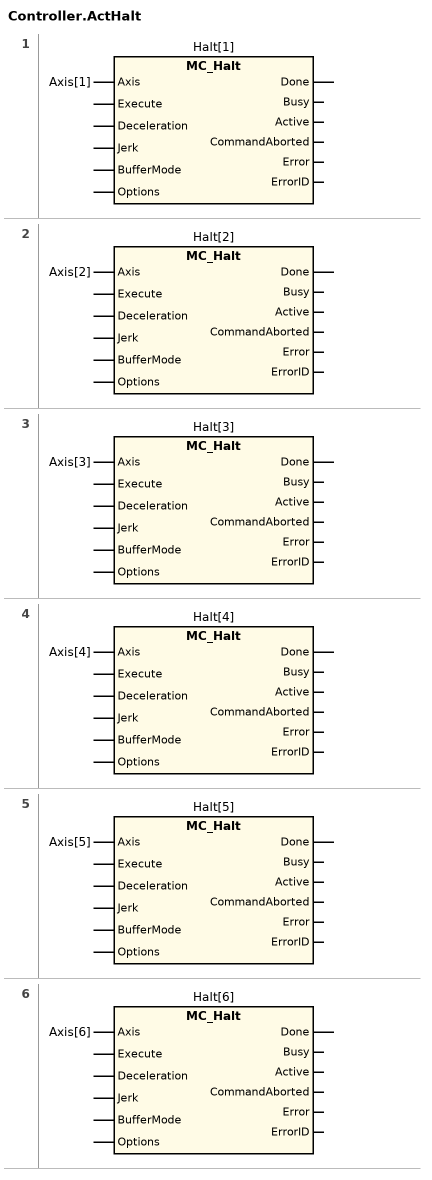
// NETWORK 1
Halt[1](Axis := Axis[1]); // MC_Halt

// NETWORK 2
Halt[2](Axis := Axis[2]); // MC_Halt

// NETWORK 3
Halt[3](Axis := Axis[3]); // MC_Halt

// NETWORK 4
Halt[4](Axis := Axis[4]); // MC_Halt

// NETWORK 5
Halt[5](Axis := Axis[5]); // MC_Halt

// NETWORK 6
Halt[6](Axis := Axis[6]); // MC_Halt
END_ACTION

ACTION ActPower:
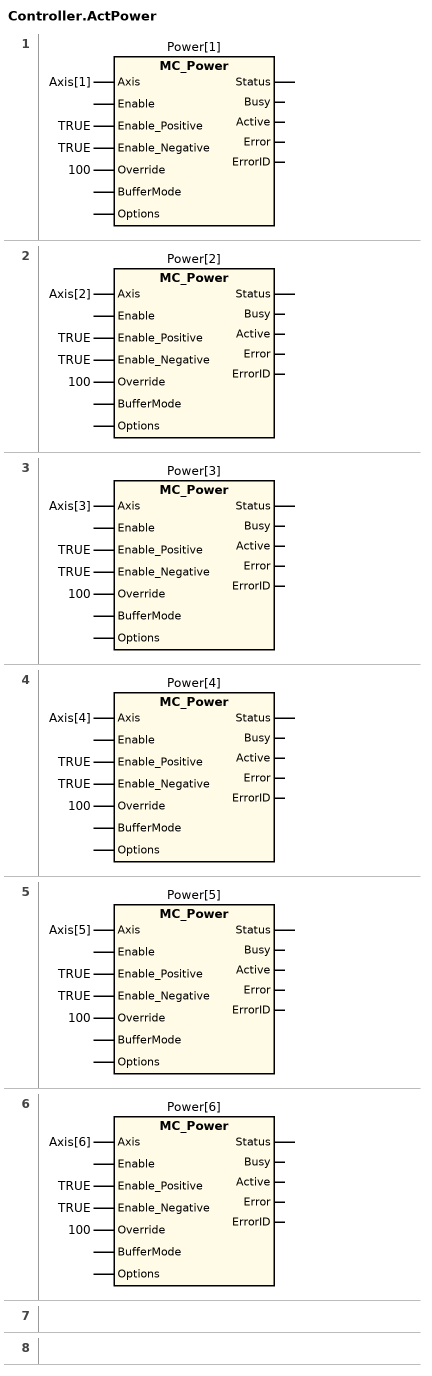
// NETWORK 1
Power[1](Axis := Axis[1], Enable_Positive := TRUE, Enable_Negative := TRUE, Override := 100); // MC_Power

// NETWORK 2
Power[2](Axis := Axis[2], Enable_Positive := TRUE, Enable_Negative := TRUE, Override := 100); // MC_Power

// NETWORK 3
Power[3](Axis := Axis[3], Enable_Positive := TRUE, Enable_Negative := TRUE, Override := 100); // MC_Power

// NETWORK 4
Power[4](Axis := Axis[4], Enable_Positive := TRUE, Enable_Negative := TRUE, Override := 100); // MC_Power

// NETWORK 5
Power[5](Axis := Axis[5], Enable_Positive := TRUE, Enable_Negative := TRUE, Override := 100); // MC_Power

// NETWORK 6
Power[6](Axis := Axis[6], Enable_Positive := TRUE, Enable_Negative := TRUE, Override := 100); // MC_Power

// NETWORK 7

// NETWORK 8
END_ACTION

ACTION ActReset:
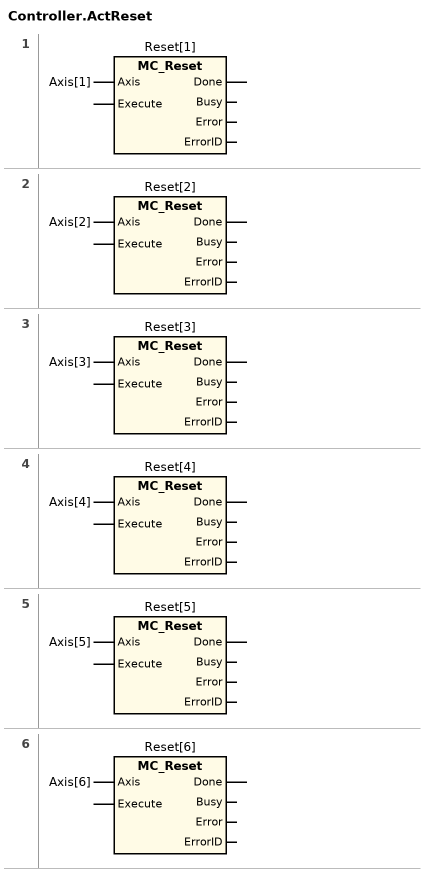
// NETWORK 1
Reset[1](Axis := Axis[1]); // MC_Reset

// NETWORK 2
Reset[2](Axis := Axis[2]); // MC_Reset

// NETWORK 3
Reset[3](Axis := Axis[3]); // MC_Reset

// NETWORK 4
Reset[4](Axis := Axis[4]); // MC_Reset

// NETWORK 5
Reset[5](Axis := Axis[5]); // MC_Reset

// NETWORK 6
Reset[6](Axis := Axis[6]); // MC_Reset
END_ACTION

ACTION ActStop:
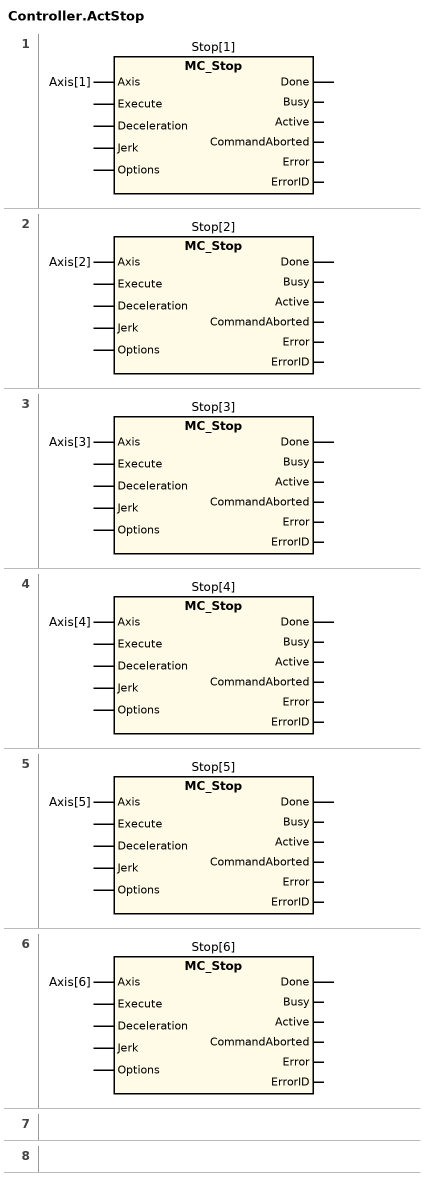
// NETWORK 1
Stop[1](Axis := Axis[1]); // MC_Stop

// NETWORK 2
Stop[2](Axis := Axis[2]); // MC_Stop

// NETWORK 3
Stop[3](Axis := Axis[3]); // MC_Stop

// NETWORK 4
Stop[4](Axis := Axis[4]); // MC_Stop

// NETWORK 5
Stop[5](Axis := Axis[5]); // MC_Stop

// NETWORK 6
Stop[6](Axis := Axis[6]); // MC_Stop

// NETWORK 7

// NETWORK 8
END_ACTION

ACTION Decider:
IF NOT state.moving AND AbsMove[1].Done AND AbsMove[2].Done AND AbsMove[3].Done AND AbsMove[4].Done  AND AbsMove[5].Done AND AbsMove[6].Done THEN
	command := E_6axis_Command.NO_COMMAND;	
END_IF

IF state.error THEN
	command := E_6Axis_Command.RESET;
END_IF

IF isHalt THEN
	command := E_6Axis_Command.HALT;
END_IF
END_ACTION

METHOD mode_Curve : BOOL

VAR_INPUT
	six_mat : ARRAY [1..6, 1..6] OF LREAL;
END_VAR

VAR_OUTPUT
	execute_fullTime : LREAL;
	coeffCopy : ARRAY [1..6, 1..6] OF LREAL;
END_VAR

VAR
	idx : DINT;
	i, j : INT;
	t : LREAL;
	temp : LREAL; // 導正係數用
	
	startAngles : ARRAY [1..6] OF LREAL;
	finalAngles : ARRAY [1..6] OF LREAL;
	pos01, pos02 : ARRAY [1..3] OF LREAL; //start and final point for calculate fulltime
	
	six_matCopy : ARRAY [1..6, 1..6] OF LREAL;
	TimeMatrix : ARRAY [1..6, 1..6] OF LREAL;
END_VAR
// Angles_mat
six_matCopy := six_mat;  // 含有角度 := 含有座標
FOR idx := 1 TO 6 DO 
	IF (idx < 3) THEN
		pos01[idx] := six_mat[idx, 1];
		pos02[idx] := six_mat[idx, 4];
	END_IF
	startAngles[idx] := six_mat[idx, 1];
	finalAngles[idx] := six_mat[idx, 4];
END_FOR
KM.Inverse(position := startAngles, degrees => startAngles);
KM.Inverse(position := finalAngles, degrees => finalAngles);
FOR idx := 1 TO 6 DO 
	six_matCopy[idx, 1] := startAngles[idx];
	six_matCopy[idx, 4] := finalAngles[idx];
END_FOR

MF.FindFullTime(pos01, pos02, 10, execute_fullTime => execute_fullTime);
t := execute_fullTime;
// Time_mat
FOR i := 1 TO 6 DO
    FOR j := 1 TO 6 DO
        CASE j OF
            1: 
                // 第一列固定為1、0、0、0、0、0
                TimeMatrix[i, j] := SEL(i = 1, 0, 1);
            2: 
                // 第二列固定為0、1、0、0、0、0
                TimeMatrix[i, j] := SEL(i = 2, 0, 1);
            3:
                // 第三列固定為0、0、2、0、0、0
                TimeMatrix[i, j] := SEL(i = 3, 0, 2);
            4:
                // 第四列公式：1 * EXPT(t, i)
                TimeMatrix[i, j] := EXPT(t, i-1);
            5:
                // 第五列公式：i * EXPT(t, i-1)
                TimeMatrix[i, j] := (i-1) * EXPT(t, i-2);
            6:
                // 第六列公式：(i * (i - 1)) * EXPT(t, i-2)
                TimeMatrix[i, j] := (i-1) * (i-2) * EXPT(t, i-3);
        END_CASE
    END_FOR
END_FOR

MF.GaussianElimination(base_mat := TimeMatrix, extend_mat := six_matCopy, temp_mat := coeffCopy, 6); //inverse 會搞壞原本的東西

FOR i := 1 TO 6 DO
	FOR j := 1 TO 3 DO
		temp := coeffCopy[i, j];
		coeffCopy[i, j] := coeffCopy[i, 7-j];
		coeffCopy[i, 7-j] := temp;
	END_FOR		
END_FOR
END_METHOD

METHOD mode_Linear : BOOL

VAR_INPUT
	six_pos : ARRAY [1..6, 1..6] OF LREAL;
END_VAR

VAR_OUTPUT
	execute_fullTime : LREAL;
	coeffCopy : ARRAY [1..6, 1..6] OF LREAL;
END_VAR

VAR
	idx : DINT;
	i, j : DINT;
	temp : LREAL; // 導正係數用

	pos01, pos02 : ARRAY [1..3] OF LREAL; //start and final point
	temp_pos : ARRAY [1..6] OF LREAL;
	temp_ang : ARRAY [1..6] OF LREAL;
	six_pos_angles : ARRAY [1..6, 1..6] OF LREAL;
	
	six_time : ARRAY [1..6, 1..6] OF LREAL;
	timeCopy : ARRAY [1..6, 1..6] OF LREAL;
	
END_VAR
// Angles_mat
FOR i := 1 TO 6 DO
	FOR j := 1 TO 6 DO
		temp_pos[j] := six_pos[i, j];
	END_FOR
	KM.Inverse(position := temp_pos, degrees => temp_ang);
	FOR j := 1 TO 6 DO
		six_pos_angles[j, i] := temp_ang[j];
	END_FOR
END_FOR

FOR idx := 1 TO 3 DO 
	pos01[idx] := six_pos[1, idx];
	pos02[idx] := six_pos[6, idx];
END_FOR
MF.FindFullTime(pos01, pos02, 10, execute_fullTime => execute_fullTime);

// Time_mat
FOR i := 1 TO 6 DO
	six_time[1, i] := 1;
	six_time[2, i] := (execute_fullTime)/5 * (i-1);
	FOR j := 3 TO 6 DO
		six_time[j, i] := EXPT(six_time[2, i], j-1);
	END_FOR
END_FOR

FOR i := 1 TO 6 DO
	FOR j := 1 TO 6 DO
		coeffCopy[i, j] := 0; // clear temp
		timeCopy[i, j] := six_time[i, j];
	END_FOR
END_FOR

MF.GaussianElimination(base_mat := timeCopy, extend_mat := six_pos_angles, temp_mat := coeffCopy, 6); //inverse 會搞壞原本的東西

FOR i := 1 TO 6 DO
	FOR j := 1 TO 3 DO
		temp := coeffCopy[i, j];
		coeffCopy[i, j] := coeffCopy[i, 7-j];
		coeffCopy[i, 7-j] := temp;
	END_FOR		
END_FOR
END_METHOD

METHOD mode_PTP : BOOL

VAR_INPUT
	angles01 : ARRAY [1..6] OF LREAL; // start position (degree)
	angles02 : ARRAY [1..6] OF LREAL; // final position (degree)
END_VAR

VAR
	idx : DINT;
	
	longest_distance : LREAL := 0;
	//time_factor : LREAL;
	execute_fullTime : LREAL := 3;
	
END_VAR
//// Execute Time
//FOR idx := 1 TO 6 DO
//	longest_distance := MAX(longest_distance, ABS(angles02[idx] - angles01[idx]));
//END_FOR
//time_factor := EXPT(30, -1); // The larger the denominator, the faster the speed
//execute_fullTime := time_factor * longest_distance;
//execute_fullTime := LREAL_TO_DINT(execute_fullTime * 1000)/1000; // Adjust Time
//IF execute_fullTime < 0.01 THEN
//	execute_fullTime := 3;
//END_IF

FOR idx := 1 TO 6 DO
	AbsMove[idx].Position := angles02[idx];
	AbsMove[idx].Velocity := ABS(angles02[idx] - Axis[idx].NcToPlc.ActPos) / execute_fullTime;
	IF AbsMove[Idx].Velocity < 0.001 THEN
		AbsMove[Idx].Velocity := 0.001;  // Module Minium Limit
	END_IF
END_FOR
END_METHOD

METHOD readAxis : BOOL

VAR
	
END_VAR
FOR idx := AXIS_MIN_IDX TO AXIS_MAX_IDX DO
	Axis[idx]();
	JointDegNow[idx] := Axis[idx].NcToPlc.ActPos;
END_FOR
KM.Forward(angles := JointDegNow, position => PositionNow);

state.powerOn := Power[1].Status AND Power[2].Status AND Power[3].Status AND Power[4].Status AND Power[5].Status AND Power[6].Status;
state.stop := Stop[1].Done AND Stop[2].Done AND Stop[3].Done AND Stop[4].Done AND Stop[5].Done AND Stop[6].Done;
state.moving := Axis[1].Status.Moving OR Axis[2].Status.Moving OR Axis[3].Status.Moving OR  Axis[4].Status.Moving OR Axis[5].Status.Moving OR Axis[6].Status.Moving;
//state.pause := NOT (state.moving OR state.stop);
state.error := Axis[1].Status.Error OR Axis[2].Status.Error OR Axis[3].Status.Error OR Axis[4].Status.Error OR Axis[5].Status.Error OR Axis[6].Status.Error;
END_METHOD

METHOD SetMotion : BOOL

VAR_INPUT
	mode : DINT;
	StartPOS : ARRAY [1..6] OF LREAL;
	FinalPOS : ARRAY [1..6] OF LREAL;
	isSIM : BOOL;
	precise : BOOL; // 專門給Homing指令使用
	
END_VAR

VAR_OUTPUT
	runTime : LREAL;
	coeffCopy : ARRAY[1..6, 1..6] OF LREAL;
END_VAR

VAR
	// PTP
	ptpAngles_01 : ARRAY [1..6] OF LREAL;
	ptpAngles_02 : ARRAY [1..6] OF LREAL;
	
	// Linear
	six_pos : ARRAY [1..6, 1..6] OF LREAL;

	
	// Curve 
	six_mat : ARRAY [1..6, 1..6] OF LREAL;
	
	// Linear & Curve
	customAngles : ARRAY [1..6] OF LREAL;  // deg & rad

	PTPMove_done : BOOL;
END_VAR


CASE mode OF
	0: // PTP
		FOR idx := AXIS_MIN_IDX TO AXIS_MAX_IDX DO
			AbsMove[idx].Execute := TRUE;
			IF NOT precise THEN
				KM.Inverse(position := StartPOS, degrees => ptpAngles_01);
				KM.Inverse(position := FinalPOS, degrees => ptpAngles_02);
				mode_PTP(ptpAngles_01, ptpAngles_02);
			ELSE
				AbsMove[idx].Position := HomeJoint[idx];
				AbsMove[idx].Velocity := 5;
			END_IF
		END_FOR		
		
		PTPMove_done := TRUE;
		FOR idx := 1 TO 6 DO
			IF NOT AbsMove[idx].Done THEN
				PTPMove_done := FALSE;
				EXIT;
			END_IF
		END_FOR
		
	1: // LINEAR
		KM.Inverse(position := FinalPOS, degrees => customAngles);
								
		FOR idx := AXIS_MIN_IDX TO AXIS_MAX_IDX DO
			ExtSwitchEn[idx].Position := customAngles[idx];
			ExtSwitchEn[idx].Execute := TRUE;
			ExtSwitchDis[idx].Execute := FALSE;
		END_FOR
		
		MF.FindForSixPoints(StartPOS, FinalPOS, six_pos => six_pos);
		mode_Linear(six_pos, coeffCopy => coeffCopy, execute_fullTime => runTime);
		
		LinearMove.Execute := TRUE;
		LinearMove.CoeffCopy := coeffCopy;
		LinearMove.RunTime := runTime;
	
	2: // CURVE
		KM.Inverse(position := FinalPOS, degrees => customAngles);
		
		FOR idx := AXIS_MIN_IDX TO AXIS_MAX_IDX DO
			ExtSwitchEn[idx].Position := customAngles[idx];
			ExtSwitchEn[idx].Execute := TRUE;
			ExtSwitchDis[idx].Execute := FALSE;
		END_FOR

		FOR idx := AXIS_MIN_IDX TO AXIS_MAX_IDX DO
			six_mat[idx, 1] :=  StartPOS[idx];
			six_mat[idx, 2] :=  StartVEL[idx];
			six_mat[idx, 3] :=  StartACC[idx];
			six_mat[idx, 4] :=  FinalPOS[idx];
			six_mat[idx, 5] :=  FinalVEL[idx];
			six_mat[idx, 6] :=  FinalACC[idx];
		END_FOR
		mode_Curve(six_mat, coeffCopy => coeffCopy, execute_fullTime => runTime);
		
		LinearMove.Execute := TRUE;
		LinearMove.CoeffCopy := coeffCopy;
		LinearMove.RunTime := runTime;
END_CASE

IF NOT isSIM AND (PTPMove_done OR LinearMove.Done) THEN
	// SetStartPosition
	IF precise THEN
		InitalPOS := HomePoint;
	ELSE

		LinearMove.Execute := FALSE;
		//running := FALSE;
		FOR idx := AXIS_MIN_IDX TO AXIS_MAX_IDX DO
			AbsMove[idx].Execute := FALSE;
			ExtSwitchEn[idx].Execute := FALSE;
			ExtSwitchDis[idx].Execute := TRUE;
		END_FOR
		InitalPOS := FinalPOS;
	END_IF
	ActExecute := FALSE;
END_IF
END_METHOD

ACTION SetStartPosition:
// IDEAL SET STARTPOSISTION
//IF NOT state.moving THEN
//	StartPosition_Now := PositionNow;
//END_IF
END_ACTION

ACTION Update_AbsMove_Motion:
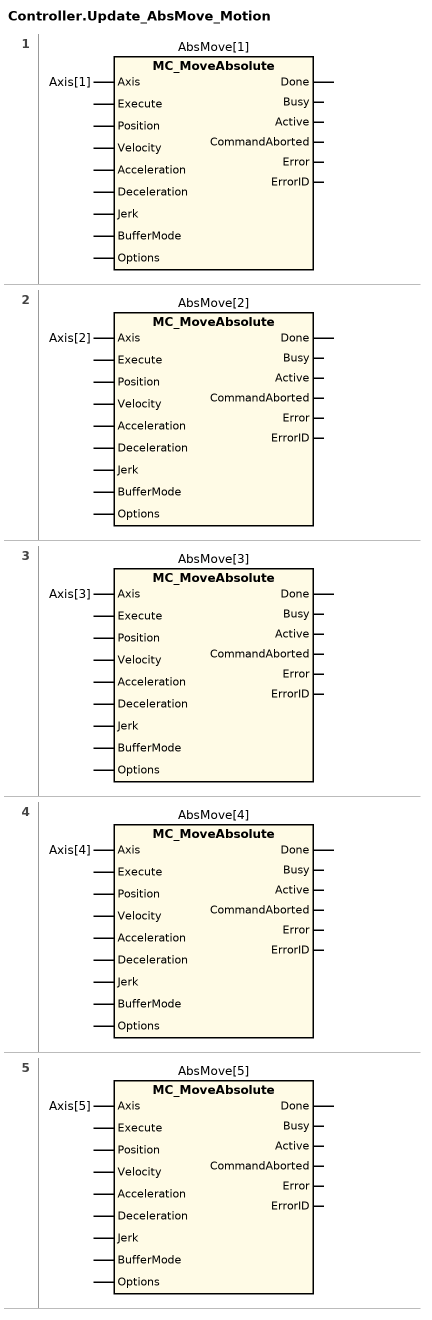
// NETWORK 1
AbsMove[1](Axis := Axis[1]); // MC_MoveAbsolute

// NETWORK 2
AbsMove[2](Axis := Axis[2]); // MC_MoveAbsolute

// NETWORK 3
AbsMove[3](Axis := Axis[3]); // MC_MoveAbsolute

// NETWORK 4
AbsMove[4](Axis := Axis[4]); // MC_MoveAbsolute

// NETWORK 5
AbsMove[5](Axis := Axis[5]); // MC_MoveAbsolute

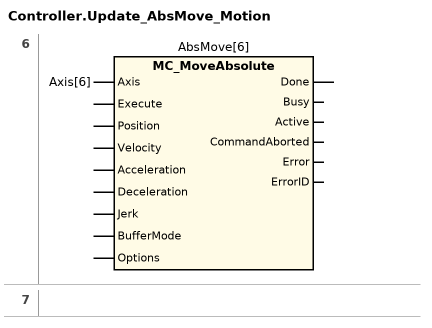
// NETWORK 6
AbsMove[6](Axis := Axis[6]); // MC_MoveAbsolute

// NETWORK 7
END_ACTION

ACTION Update_Custom_Motion:
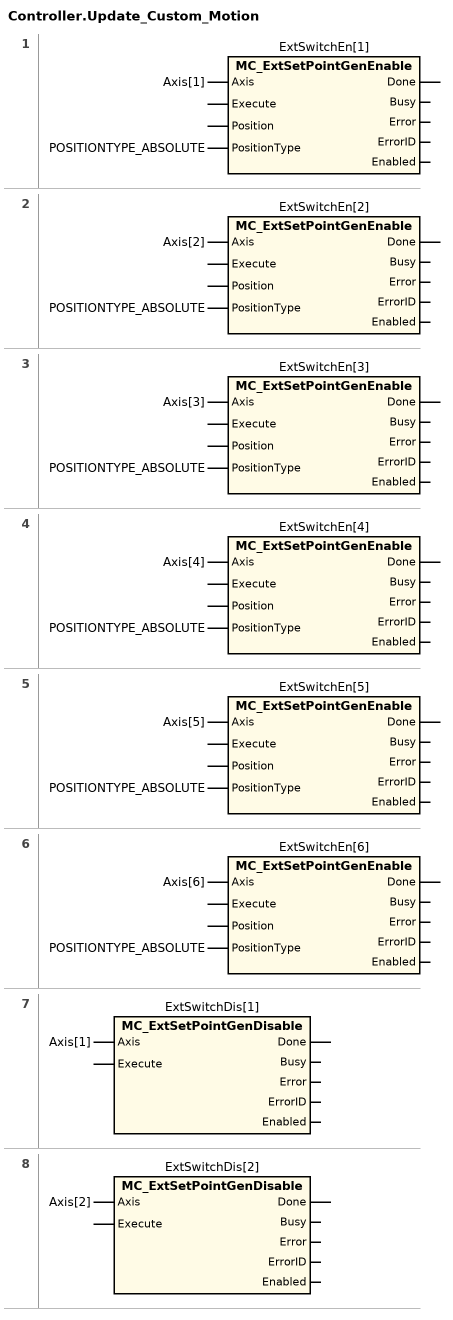
// NETWORK 1
ExtSwitchEn[1](Axis := Axis[1], PositionType := POSITIONTYPE_ABSOLUTE); // MC_ExtSetPointGenEnable

// NETWORK 2
ExtSwitchEn[2](Axis := Axis[2], PositionType := POSITIONTYPE_ABSOLUTE); // MC_ExtSetPointGenEnable

// NETWORK 3
ExtSwitchEn[3](Axis := Axis[3], PositionType := POSITIONTYPE_ABSOLUTE); // MC_ExtSetPointGenEnable

// NETWORK 4
ExtSwitchEn[4](Axis := Axis[4], PositionType := POSITIONTYPE_ABSOLUTE); // MC_ExtSetPointGenEnable

// NETWORK 5
ExtSwitchEn[5](Axis := Axis[5], PositionType := POSITIONTYPE_ABSOLUTE); // MC_ExtSetPointGenEnable

// NETWORK 6
ExtSwitchEn[6](Axis := Axis[6], PositionType := POSITIONTYPE_ABSOLUTE); // MC_ExtSetPointGenEnable

// NETWORK 7
ExtSwitchDis[1](Axis := Axis[1]); // MC_ExtSetPointGenDisable

// NETWORK 8
ExtSwitchDis[2](Axis := Axis[2]); // MC_ExtSetPointGenDisable

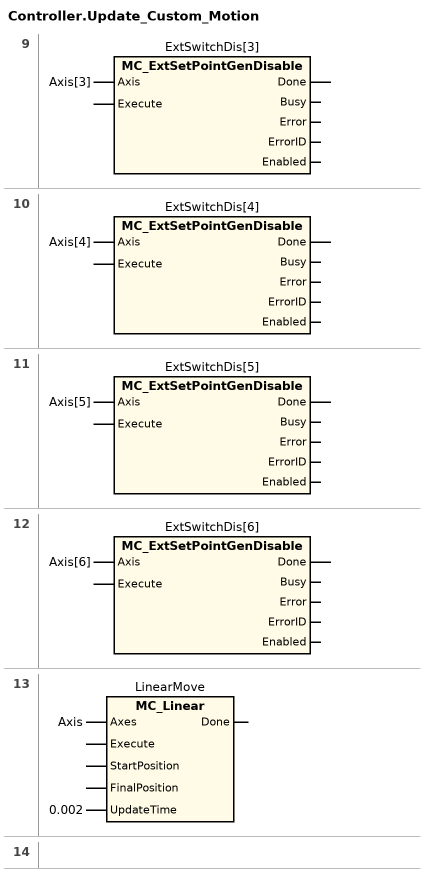
// NETWORK 9
ExtSwitchDis[3](Axis := Axis[3]); // MC_ExtSetPointGenDisable

// NETWORK 10
ExtSwitchDis[4](Axis := Axis[4]); // MC_ExtSetPointGenDisable

// NETWORK 11
ExtSwitchDis[5](Axis := Axis[5]); // MC_ExtSetPointGenDisable

// NETWORK 12
ExtSwitchDis[6](Axis := Axis[6]); // MC_ExtSetPointGenDisable

// NETWORK 13
LinearMove(Axes := Axis, UpdateTime := 0.002); // MC_Linear

// NETWORK 14
END_ACTION

END_FUNCTION_BLOCK

// ---- POUs/Buffer.TcPOU
FUNCTION_BLOCK Buffer

VAR CONSTANT
	AxesMaxAmount : USINT := 6;
	PosMaxAmount : USINT := 10;
END_VAR

VAR
	bInit : BOOL := TRUE;
	POS_STORAGE : ARRAY [1..PosMaxAmount] OF ARRAY [1..AxesMaxAmount] OF LREAL;
	InCommand : Motion_Command_Input;
END_VAR



InCommand.StartPos := InCommand.StartPOS;

END_FUNCTION_BLOCK

// ---- POUs/Kinematics.TcPOU
FUNCTION_BLOCK PUBLIC Kinematics

VAR CONSTANT
	L1 : ARRAY[1..3] OF LREAL := [0, 0, 289];    
	L2 : ARRAY[1..3] OF LREAL := [105, 0, 200];
	L3 : ARRAY[1..3] OF LREAL := [0, 0, 280];
	L4 : ARRAY[1.   .3] OF LREAL := [146, 0, 65];
	L5 : ARRAY[1..3] OF LREAL := [174, 0, 0];
	L6 : ARRAY[1..3] OF LREAL := [140, 0, 0];
	
	L35 : LREAL := SQRT(EXPT(L4[3], 2) + EXPT(L4[1] + L5[1], 2)); // L35 = The Length of J3 to J5
	L25_MAX : LREAL := L3[3] + L35;
	L25_MIN : LREAL := ABS(L3[3] - L35);
	
	
END_VAR

VAR
	// if only use Forward or Inverse Kinematics
	TestPOS : ARRAY[1..6] OF LREAL := [330, -150, 280, -42, 0, 45];
	TestJOINT : ARRAY[1..6] OF LREAL := [0, 45, 45, 0, -90, 49.5];
	
	angles : ARRAY[1..6] OF LREAL; 
	pos : ARRAY[1..6] OF LREAL; 
END_VAR

Inverse(position := TestPOS, degrees => angles);
Forward(angles := TestJOINT, position => pos);

METHOD PUBLIC _atan : LREAL
VAR_INPUT
	y : LREAL;
	x : LREAL;
END_VAR
IF x > 0 THEN
	_atan := ATAN(y/x);
ELSIF x = 0 THEN
	IF y = 0 THEN
		_atan := 0;
	ELSIF y > 0 THEN
		_atan := PI/2;
	ELSIF y < 0 THEN
		_atan := -PI/2;
	END_IF
ELSE
	IF y >= 0 THEN
		_atan := ATAN(y / x) + PI;
	ELSE
		_atan := ATAN(y / x) - PI;
	END_IF
END_IF
END_METHOD

METHOD PUBLIC _d2r : LREAL

VAR_INPUT
	degrees : LREAL;
END_VAR
_d2r := degrees * PI / 180.0;
END_METHOD

METHOD _matrixMultipl : LREAL
VAR_INPUT
	A : ARRAY[1..3, 1..3] OF LREAL;
	B : ARRAY[1..3, 1..3] OF LREAL;
END_VAR

VAR_OUTPUT
	C : ARRAY[1..3, 1..3] OF LREAL;
END_VAR

VAR 
	i: DINT;   // row
	j : DINT;  // col
END_VAR
FOR i := 1 TO 3 DO
	FOR j := 1 TO 3 DO
		C[i, j] := A[i, 1] * B[1, j] + A[i, 2] * B[2, j] + A[i, 3] * B[3, j];
	END_FOR
END_FOR
END_METHOD

METHOD PUBLIC _r2d : LREAL

VAR_INPUT
	radians : LREAL;
END_VAR
_r2d := radians * 180.0 / PI;
END_METHOD

METHOD PUBLIC _rodLength : LREAL
VAR_INPUT
	xyz : ARRAY[1..3] OF LREAL;
END_VAR
_rodLength := EXPT(xyz[1], 2) + EXPT(xyz[1], 2) + EXPT(xyz[1], 2);
IF _rodLength <= 0 THEN
	_rodLength := 100;
END_IF
_rodLength := SQRT(_rodLength);
END_METHOD

METHOD PUBLIC _sign : LREAL
VAR_INPUT
	number : LREAL;
END_VAR
IF number > 0 THEN
	_sign := 1;
ELSIF number < 0 THEN
	_sign := -1;
ELSE
	_sign := 0;
END_IF
END_METHOD

METHOD Forward : BOOL

VAR_INPUT
	angles : ARRAY[1..6] OF LREAL; // joints' angle in radians
END_VAR

VAR_OUTPUT
	// position : [x, y, z, r, p, y]
	position : ARRAY[1..6] OF LREAL; 
END_VAR

VAR
	idx : int;

	c1 : LREAL;
	c2 : LREAL;
	c4 : LREAL;
	c5 : LREAL;
	c6 : LREAL;
	c23 : LREAL;
	s1 : LREAL;
	s2 : LREAL;
	s4 : LREAL;
	s5 : LREAL;
	s6 : LREAL;
	s23 : LREAL;
	
	// Position repeat value
	L05_XY : LREAL;
	
	// Part of the fixed frame rotation matrix element(X->Y->Z) => R = Rz*Ry*Rx
	r11 : LREAL;  // cos(Ry)*cos(Rz)
	r12 : LREAL;  // sin(Rx)*sin(Ry)*cos(Rz) - cos(Rx)*sin(Rz)
	r21 : LREAL;  // cos(Ry)*sin(Rz)
	r22 : LREAL;  // cos(Rx)*cos(Rz) + sin(Rx)*sin(Ry)*sin(Rz)
	r31 : LREAL;  // -sin(Ry)
	r32 : LREAL;  // cos(Ry)*sin(Rx)
	r33 : LREAL;  // cos(Ry)*cos(Rx)
END_VAR
// The lazy implementation is directly multipling 6 of 4x4 transform matrices based on
// world frame, and the below program is simplified result which is derived from
// TF06 := TF01 * TF12 * TF23 * TF34 * TF45 * TF56
// where the position vector of each transform matrix is refrenced by link vector, and the rotation
// matrices are rotate along specific world frame axis in the following order(TF01 to TF06)
// R01(Z) -> R12(Y) -> R23(Y) -> R34(X) -> R45(Y) -> R56(X)
FOR idx := 1 TO 6 DO
	angles[idx] := _d2r(angles[idx]);
END_FOR


c1 := COS(angles[1]);
c2 := COS(angles[2]);
c4 := COS(angles[4]);
c5 := COS(angles[5]);
c6 := COS(angles[6]);
c23 := COS(angles[2] + angles[3]);

s1 := SIN(angles[1]);
s2 := SIN(angles[2]);
s4 := SIN(angles[4]);
s5 := SIN(angles[5]);
s6 := SIN(angles[6]);
s23 := SIN(angles[2] + angles[3]);

// Position
L05_XY := L2[1] + L3[3]*s2 + L4[3]*s23 + (L4[1] + L5[1])*c23;
position[1] := c1*L05_XY + L6[1]*(c5*c1*c23 - s5*(s1*s4 + c1*s23*c4));
position[2] := s1*L05_XY + L6[1]*s1*(c23*c5 - s23*c4*s5) + L6[1]*c1*s4*s5;		
position[3] := L1[3] + L2[3] + L3[3]*c2 + L4[3]*c23 - (L4[1] + L5[1])*s23 - L6[1]*(s23*c5 + c23*c4*s5);

// Rotation matrix to fixed frame rotation angels
r31 := -s23*c5 - c23*c4*s5;
IF ABS(r31) <> 1.0 THEN  // Pitch angle(Ry) not equal to +-pi/2
	r11 := c1*c23*c5 - s5*(s1*s4 + c1*s23*c4);
	r21 := s1*c23*c5 + s5*(c1*s4 - s1*s23*c4);
	r32 := c23*s4*c6 - s6*(s23*s5 - c23*c4*c5);
	r33 := -c23*s4*s6 - c6*(s23*s5 - c23*c4*c5);
	
	position[4] := _atan(r32, r33);
	position[6] := _atan(r21, r11);
	IF COS(position[6]) = 0.0 THEN
		position[5] := _atan(-r31, r21/SIN(position[6]));
	ELSE
		position[5] := _atan(-r31, r11/COS(position[6]));
	END_IF
ELSE  // Gimbal lock when picth angle(Ry) is equal to +-pi/2
	r12 := -c6*(s1*c4 - c1*s23*s4) + s6*(c1*c23*s5 + c5*(s1*s4 + c1*s23*c4));
	r22 :=  c6*(c1*c4 + s1*s23*s4) + s6*(s1*c23*s5 - c5*(c1*s4 - s1*s23*c4));

	position[4] := 0;
    position[5] := _atan(-r31, 0);
    position[6] := _atan(-r12, r22);
END_IF

FOR idx := 4 TO 6 DO
	position[idx] := _r2d(position[idx]);
END_FOR
END_METHOD

METHOD PUBLIC Inverse : BOOL

VAR_INPUT
	// position : [x, y, z, r, p, y]
	position : ARRAY[1..6] OF LREAL; 
END_VAR

VAR_OUTPUT
	degrees : ARRAY[1..6] OF LREAL;  // joints' angle(degree)
	radians : ARRAY[1..6] OF LREAL;  // joints' angle(radians)
END_VAR
	
VAR
	idx : INT;
	
	xyz : ARRAY[1..3] OF LREAL;  // position(mm)
	rpy : ARRAY[1..3] OF LREAL;  // rotation(degree)
	angles : ARRAY[1..6] OF LREAL;  // joints' angle(degree)
	
	R06 : ARRAY[1..3, 1..3] OF LREAL;
	R03_T : ARRAY[1..3, 1..3] OF LREAL;
	pos_J5 : ARRAY[1..3] OF LREAL; 
	
	c1 : LREAL;
	s1 : LREAL;
	pos_J2 : ARRAY[1..3] OF LREAL; 
	
	L25_square : LREAL := 0; 
	phi : LREAL;
	
	c23 : LREAL;
	s23 : LREAL;
	
	R36 : ARRAY[1..3, 1..3] OF LREAL;
	
	atan2: INT;
	
	
END_VAR
FOR idx := 1 TO 3 DO
	xyz[idx] := position[idx];
	rpy[idx] := _d2r(position[idx + 3]);
END_FOR

pos_J5[1] := xyz[1] - L6[1] * COS(rpy[2]) * COS(rpy[3]);
pos_J5[2] := xyz[2] - L6[1] * COS(rpy[2]) * SIN(rpy[3]);
pos_J5[3] := xyz[3] - L6[1] * SIN(rpy[2]) * -1;

radians[1] := _atan(y := pos_J5[2], x := pos_J5[1]);
c1 := COS(radians[1]);
s1 := SIN(radians[1]);

pos_J2[1] := L2[1] * c1;
pos_J2[2] := L2[1] * s1;
pos_J2[3] := L1[3] + L2[3];

FOR idx := 1 TO 3 DO
	L25_square := L25_square + EXPT(pos_J5[idx] - pos_J2[idx], 2);
END_FOR

IF L25_square > EXPT(L25_MAX, 2) OR L25_square < EXPT(L25_MIN, 2) THEN
	inverse := FALSE;
	RETURN;
END_IF

phi := ACOS((pos_J5[3] - pos_J2[3]) / SQRT(L25_square));
radians[2] := phi
			 - ACOS((EXPT(L3[3], 2) + L25_square - EXPT(L35, 2)) / (2 * SQRT(L25_square) * L3[3]));
radians[3] := PI/2
             - ACOS((EXPT(L3[3], 2) + EXPT(L35, 2) - L25_square) / (2 * L3[3] * L35) )
			 + ATAN(L4[3] / (L4[1] + L5[1]));

// find R36, R06 = R03 * R36
// known R06、 R03, R is meaning Rotation matrix
// inv(R03) * R6 = transpose(R03) * R06
c23 := COS(radians[2] + radians[3]);
s23 := SIN(radians[2] + radians[3]);

R06[1, 1] := COS(rpy[2]) * COS(rpy[3]);
R06[1, 2] := SIN(rpy[1]) * SIN(rpy[2]) * COS(rpy[3]) - COS(rpy[1]) * SIN(rpy[3]);
R06[1, 3] := COS(rpy[1]) * SIN(rpy[2]) * COS(rpy[3]) + SIN(rpy[1]) * SIN(rpy[3]);
R06[2, 1] := COS(rpy[2]) * SIN(rpy[3]);
R06[2, 2] := SIN(rpy[1]) * SIN(rpy[2]) * SIN(rpy[3]) + COS(rpy[1]) * COS(rpy[3]);
R06[2, 3] := COS(rpy[1]) * SIN(rpy[2]) * SIN(rpy[3]) - SIN(rpy[1]) * COS(rpy[3]);
R06[3, 1] := SIN(rpy[2]) * -1;
R06[3, 2] := SIN(rpy[1]) * COS(rpy[2]);
R06[3, 3] := COS(rpy[1]) * COS(rpy[2]);

R03_T[1, 1] := c1 * c23;
R03_T[1, 2] := s1 * c23;
R03_T[1, 3] := -s23;
R03_T[2, 1] := -s1;
R03_T[2, 2] := c1;
R03_T[2, 3] := 0;
R03_T[3, 1] := c1 * s23;
R03_T[3, 2] := s1 * s23;
R03_T[3, 3] := c23;
_matrixMultipl(A := R03_T, B := R06, C => R36);
radians[4] := _atan(R36[2, 1], -R36[3, 1]);
radians[6] := _atan(R36[1, 2], R36[1, 3]);
radians[5] := _atan(R36[1, 3]/COS(radians[6]), R36[1,1]);

IF ABS(radians[4]) > PI/2 THEN
	radians[4] := radians[4]  - _sign(radians[4]) * PI;
	radians[5] := -radians[5];
	radians[6] := radians[6] - _sign(radians[6]) * PI;
END_IF

//判斷是否在工作範圍
IF _d2r(-180) <= radians[1] AND radians[1] <= _d2r(180) AND
   _d2r(-57 ) <= radians[2] AND radians[2] <= _d2r(120) AND
   _d2r(-125) <= radians[3] AND radians[3] <= _d2r(55 ) AND
   _d2r(-180) <= radians[4] AND radians[4] <= _d2r(180) AND
   _d2r(-124) <= radians[5] AND radians[5] <= _d2r(115) AND
   _d2r(-180) <= radians[6] AND radians[6] <= _d2r(180) THEN
   
	FOR idx := 1 TO 6 DO
		degrees[idx] := _r2d(radians[idx]);
		radians[idx] := radians[idx];
	END_FOR
ELSE
	
	isHalt := TRUE;
	RETURN;
END_IF
END_METHOD

END_FUNCTION_BLOCK

// ---- POUs/MathFunc.TcPOU
FUNCTION_BLOCK MathFunc

METHOD Factorial : LREAL
VAR_INPUT
    n : INT;
END_VAR

VAR
	i : INT;
    result: INT := 1;
    
END_VAR
FOR i := 1 TO n DO
    result := result * i;
END_FOR

Factorial := result;
END_METHOD

METHOD FindForSixPoints : BOOL

VAR_INPUT
	start_pos : ARRAY [1..6] OF LREAL;
	final_pos : ARRAY [1..6] OF LREAL;
END_VAR

VAR_OUTPUT
	six_pos : ARRAY [1..6, 1..6] OF LREAL;
END_VAR

VAR
	i, j : DINT;
	delta : ARRAY[1..6] OF LREAL;
	section : ARRAY[1..5] OF LREAL;
	weight : ARRAY[1..5] OF LREAL := [15, 21, 25.5, 25, 13.5];
END_VAR
FOR i := 1 TO 6 DO
	delta[i] := final_pos[i] - start_pos[i];
	FOR j := 1 TO 5 DO
		section[j] := delta[i] * weight[j] / 100;
	END_FOR
	six_pos[1, i] := start_pos[i];
	FOR j := 2 TO 6 DO
		six_pos[j, i] := six_pos[j - 1, i] + section[j - 1];
	END_FOR		
END_FOR
END_METHOD

METHOD FindFullTime : BOOL

VAR_INPUT
	pos01 : ARRAY [1..3] OF LREAL;
	pos02 : ARRAY [1..3] OF LREAL;
	time_factor : LREAL;
END_VAR

VAR_OUTPUT
	execute_fullTime : LREAL;
END_VAR

VAR
	longest_distance : LREAL;
END_VAR
longest_distance := SQRT(EXPT(pos02[1] - pos01[1], 2) + EXPT(pos02[2] - pos01[2], 2) + EXPT(pos02[3] - pos01[3], 2)); 
execute_fullTime := EXPT(time_factor, -1) * longest_distance;

//fix time proble
execute_fullTime := LREAL_TO_DINT(execute_fullTime * EXPT(10, 7))/EXPT(10, 7);
END_METHOD

METHOD GaussianElimination

// n-order trajectory curve fitting
VAR_IN_OUT
	base_mat : ARRAY[*, *] OF LREAL;    // 6 of time-related function(Assume t0 at last row)
	extend_mat : ARRAY[*, *] OF LREAL;  // target(XYZRPY) on corresponding time
	temp_mat : ARRAY[*, *] OF LREAL;  	// 暫存矩陣(放單位矩陣跟反矩陣)
END_VAR

VAR_INPUT
	order : INT;
END_VAR

VAR
	n : INT;
	row : INT;
	column : INT;
	gain : LREAL;
	temp : LREAL;
	base_mat_Copy : ARRAY [1..6] OF ARRAY [1..6] OF LREAL;
END_VAR
FOR row := 1 TO order DO
	FOR column := 1 TO order DO
		base_mat_Copy[row][column] := base_mat[row, column];
	END_FOR
END_FOR
// Create a unit
FOR row := 1 TO order DO
	FOR column := 1 TO order DO
		IF row = column THEN
			temp_mat[row, column] := 1;
		ELSE
			temp_mat[row, column] := 0;
		END_IF
	END_FOR
END_FOR

// Lower triangle to zeros
FOR n := 1 TO order DO
	FOR row := n+1 TO order DO
		gain := base_mat[row, n] / base_mat[n, n];
		// Elimination
		FOR column := 1 TO order DO
			base_mat[row, column] := base_mat[row, column] - gain * base_mat[n, column];
			// The matrix shape is exacly the same as base_mat
			temp_mat[row, column] := temp_mat[row, column] - gain * temp_mat[n, column];
		END_FOR
	END_FOR
END_FOR

// Upper triangle to zeros
FOR n := order TO 1 BY -1 DO
	FOR row := n-1 TO 1 BY -1 DO
		gain := base_mat[row, n] / base_mat[n, n];
		// Elimination
		FOR column := order TO 1 BY -1 DO
			base_mat[row, column] := base_mat[row, column] - gain * base_mat[n, column];
			// The matrix shape is exacly the same as base_mat
			temp_mat[row, column] := temp_mat[row, column] - gain * temp_mat[n, column];
		END_FOR
	END_FOR
END_FOR

// Solve equation
FOR row := 1 TO 6 DO
	FOR column := 1 TO 6 DO
		temp_mat[row, column] := temp_mat[row, column] / base_mat[row, row];
		//Round(num1 := temp_mat[row, column], n := 2, num2 => temp_mat[row, column]);
	END_FOR
END_FOR
MultiplyByMatrix(A := extend_mat, B := temp_mat, C := base_mat, n := 6);

// Switch the name of matrix
FOR row := 1 TO order DO
	FOR column := 1 TO order DO
		temp := temp_mat[row, column];
		temp_mat[row, column] := base_mat[row, column];
		base_mat[row, column] := temp;
	END_FOR		
END_FOR
END_METHOD

METHOD MultiplyByMatrix : BOOL

VAR_IN_OUT
	A : ARRAY[*, *] OF LREAL;
	B : ARRAY[*, *] OF LREAL;
	C : ARRAY[*, *] OF LREAL;
END_VAR

VAR_INPUT
	n : INT;
END_VAR

VAR 
	i: DINT;   // row
	j : DINT;  // col
	k : Dint;  // order
END_VAR
FOR i := 1 TO n DO
	FOR j := 1 TO n DO
		C[i, j] := 0;
	END_FOR
END_FOR

FOR i := 1 TO n DO
	FOR j := 1 TO n DO
		FOR k := 1 TO n DO
			C[i, j] := C[i, j] + A[i, k] * B[k, j];
			//Round(num1 := C[i, j], n := 5, num2 => C[i, j]);
		END_FOR
	END_FOR
END_FOR
END_METHOD

METHOD Round : BOOL
VAR_INPUT
	num1 : LREAL;
	n : INT;
END_VAR

VAR_OUTPUT
	num2 : lreal;
END_VAR
num2 := LREAL_TO_DINT(num1 * EXPT(10, n) ) / EXPT(10, n);
END_METHOD

METHOD VectorMotionPOS : BOOL

VAR_IN_OUT
	POS : ARRAY [AXIS_MIN_IDX..AXIS_MAX_IDX] OF LREAL;
END_VAR

VAR_INPUT
	Direcation : LREAL;
	Path_Motion_Displace : LREAL;
END_VAR
IF Direcation = 1 THEN
	POS[1] := POS[1] + Path_Motion_Displace;
ELSIF Direcation = 2 THEN
	POS[2] := POS[2] + Path_Motion_Displace;
ELSIF Direcation = 3 THEN
	POS[3] := POS[3] + Path_Motion_Displace;
ELSIF Direcation = 4 THEN
	POS[1] := POS[1] + Path_Motion_Displace * 0.5 * EXPT(2, 0.5);
	POS[2] := POS[2] + Path_Motion_Displace * 0.5 * EXPT(2, 0.5);
ELSIF Direcation = 5 THEN
	POS[1] := POS[1] + Path_Motion_Displace * 0.5 * EXPT(2, 0.5);
	POS[2] := POS[2] - Path_Motion_Displace * 0.5 * EXPT(2, 0.5);
END_IF
END_METHOD

END_FUNCTION_BLOCK

// ---- POUs/MC_Linear.TcPOU
FUNCTION_BLOCK MC_Linear

VAR CONSTANT
	AXIS_MIN_IDX : USINT := 1;
	AXIS_MAX_IDX : USINT := 6;
END_VAR

VAR_IN_OUT
	Axes : ARRAY[AXIS_MIN_IDX..AXIS_MAX_IDX] OF AXIS_REF;
	
END_VAR

VAR_INPUT
	Execute : BOOL;
	CoeffCopy : ARRAY[1..6, 1..6] OF LREAL; 
	RunTime : LREAL;
	UpdateTime : LREAL;
END_VAR

VAR_OUTPUT
	Done : BOOL;
END_VAR

VAR
	idx : DINT;
	timer : LREAL;
	lastExecute : BOOL;
	pos : LREAL;
	vel : LREAL;
	acc : LREAL;
	direction : DINT;
	RunTimeCopy : LREAL;
	UpdateTimeCopy : LREAL;
END_VAR

IF NOT Execute THEN
	Done := FALSE;
	lastExecute := Execute;
	RETURN;
END_IF

IF NOT lastExecute THEN
	RunTimeCopy := RunTime;
	updateTimeCopy := UpdateTime;
	timer := 0;
END_IF
lastExecute := Execute;

FOR idx := 1 TO 6 DO
	pos := CoeffCopy[idx, 1]*EXPT(timer, 5) + CoeffCopy[idx, 2]*EXPT(timer, 4)	
		+ CoeffCopy[idx, 3]*EXPT(timer, 3) + CoeffCopy[idx, 4]*EXPT(timer, 2) 
		+ CoeffCopy[idx, 5]*EXPT(timer, 1) + CoeffCopy[idx, 6]*EXPT(timer, 0);
								  
	vel := CoeffCopy[idx, 1]*5*EXPT(timer, 4) + CoeffCopy[idx, 2]*4*EXPT(timer, 3)
		+ CoeffCopy[idx, 3]*3*EXPT(timer, 2) + CoeffCopy[idx, 4]*2*EXPT(timer, 1)
		+ CoeffCopy[idx, 5]*1*EXPT(timer, 0);
		 
	acc := CoeffCopy[idx, 1]*20*EXPT(timer, 3) + CoeffCopy[idx, 2]*12*EXPT(timer, 2)
		+ CoeffCopy[idx, 3]*6*EXPT(timer, 1) + CoeffCopy[idx, 4]*2*EXPT(timer, 0);
		
	IF vel = 0 AND acc = 0 THEN
		direction := 0;	(* stand still *)
	ELSIF vel >= 0 THEN
		direction := 1;	(* positive motion *)
	ELSE
		direction := -1;  (* negative motion *)
	END_IF
	
	IF timer >= runTimeCopy THEN
		vel := 0;
		acc := 0;
		direction := 0;
		Done := TRUE;
	END_IF

	MC_ExtSetPointGenFeed(
		Position := pos,
		Velocity := vel,
		Acceleration := acc,
		Direction := direction,
		Axis := Axes[idx]);
END_FOR

IF NOT Done THEN
	timer := timer + updateTimeCopy;
END_IF

END_FUNCTION_BLOCK

// ---- POUs/Airbus_TCP/Serialize.TcPOU
FUNCTION_BLOCK Serialize

VAR_INPUT
	a : BYTE;
	b : LREAL;
	c : ARRAY[1..6, 1..6] OF LREAL;
END_VAR

VAR_OUTPUT
	sendbuffer : ARRAY[0..1023] OF BYTE;
END_VAR

VAR
	i, j : DINT;
	offset : UDINT := 0;
END_VAR

offset := 0;
MEMCPY(ADR(sendbuffer[offset]), ADR(a), SIZEOF(a));

offset := offset + SIZEOF(a);
MEMCPY(ADR(sendbuffer[offset]), ADR(b), SIZEOF(b));

offset := offset + SIZEOF(b);
FOR i := 1 TO 6 DO
	FOR j := 1 TO 6 DO
		MEMCPY(ADR(sendbuffer[offset]), ADR(c[i,j]), SIZEOF(c[i,j]));
		offset := offset + SIZEOF(b);
	END_FOR
END_FOR

END_FUNCTION_BLOCK

// ---- POUs/Airbus_TCP/Deserialize.TcPOU
FUNCTION_BLOCK Deserialize

VAR_INPUT
	Recvbuffer : ARRAY[0..1023] OF BYTE;
END_VAR

VAR_OUTPUT
	a : BYTE;
	b : DINT;
	c : ARRAY[1..6] OF LREAL;
END_VAR

VAR
	idx : DINT;
	offset : DINT := 0;
END_VAR

offset := 0;
MEMCPY(ADR(a), ADR(Recvbuffer[offset]), SIZEOF(a));

offset := offset + SIZEOF(a);
MEMCPY(ADR(b), ADR(Recvbuffer[offset]), SIZEOF(b));

offset := offset + SIZEOF(b);
FOR idx := 1 TO 6 DO
	MEMCPY(ADR(c[idx]), ADR(RecvBuffer[offset]), SIZEOF(c[idx]));
    offset := offset + SIZEOF(c[idx]);
END_FOR

END_FUNCTION_BLOCK

// ---- POUs/Airbus_TCP/FB_TCPClient.TcPOU
FUNCTION_BLOCK FB_TCPClient

VAR_INPUT
	sRemoteHost: T_IPv4Addr;
	nRemotePort: UDINT;
	sSendData: ARRAY[0..1023] OF BYTE;;	
	bStartCommunication: BOOL;
	tCycleTimeSend: TIME;
	bSendTrigger : BOOL;
END_VAR

VAR_OUTPUT
	bConnected: BOOL;
	sReceivedData: ARRAY[0..1023] OF BYTE;
	nErrorID: UDINT;
	bError: BOOL;
	bBusy: BOOL;
END_VAR

VAR
	iState: INT;
	fbSocketConnect: FB_SocketConnect;
	fbSocketSend: FB_SocketSend;
	deserialize: deserialize;
	fbSocketClose: FB_SocketClose;
	fbSocketReceive: FB_SocketReceive;
	hSocket: T_HSOCKET;

	fbTimer: TON;
	nRecBytes: UDINT;
	bExecuteSocketSend: BOOL;
	RTrig: R_TRIG;
	buffer : UDINT;
END_VAR

CASE iState OF
	0:	// Init State
		fbSocketConnect(bExecute := FALSE); 
		fbSocketSend(bExecute := FALSE); 
		fbSocketReceive(bExecute := FALSE);
		fbSocketClose(bExecute := FALSE); 
		bConnected := FALSE; 
		bBusy := FALSE;
		IF bStartCommunication = TRUE THEN									// Start communication manually 
			iState := iState + 10;
			bBusy := TRUE;
			bError := FALSE;
		END_IF
	
	10:	// Connect Server
		fbSocketConnect(													// Open connection to server
			sSrvNetId:= '', 
			sRemoteHost:= sRemoteHost, 
			nRemotePort:= nRemotePort, 
			bExecute:= TRUE, 
			tTimeout:= T#4S, 
			bBusy=> , 
			bError=> bError, 
			nErrId=> nErrorID, 
			hSocket=> hSocket);
	
		IF hSocket.handle <> 0 AND NOT (fbSocketConnect.bBusy) THEN			// Handle is created
			bConnected := TRUE; 
			iState :=iState + 5;
		ELSIF bError THEN
			iState := 0; 	
		END_IF
		
		
	15:																		// StartCommunication
		IF (tCycleTimeSend <> T#0MS) THEN									// Send data cyclically
			fbTimer(IN:= NOT fbTimer.Q, PT:= tCycleTimeSend, Q=> , ET=> );		
		END_IF
		RTrig(CLK:= bSendTrigger, Q=> );									// SendData on manuel trigger
		
		fbSocketSend(														// Send Data
			sSrvNetId:= '', 
			hSocket:= hSocket, 
			cbLen:= SIZEOF(sSendData), 
			pSrc:= ADR(sSendData), 
			bExecute:= (fbTimer.Q OR RTrig.Q), 
			tTimeout:= T#2S, 
			bError=> bError, 
			nErrId=> nErrorID, 
			nErrId=> );
	
		fbSocketReceive(													// ReceiveData
			sSrvNetId:= '', 
			hSocket:= hSocket, 
			cbLen:= SIZEOF(sReceivedData), 
			pDest:= ADR(sReceivedData), 
			bExecute:= true, 
			tTimeout:= T#3S, 
			bBusy=> , 
			bError=> bError, 
			nErrId=> nErrorID, 
			nRecBytes=> nRecBytes);
	
		IF NOT fbSocketReceive.bBusy THEN									// Check cyclically for new data
			fbSocketReceive(bExecute := FALSE);
		END_IF						
		IF NOT bStartCommunication OR bError THEN							// Close connection in case of error or manual communication stop
			iState := 20;
		END_IF
	20: 
		fbSocketClose(														// Close connection
			sSrvNetId:= '', 
			hSocket:= hSocket, 
			bExecute:= TRUE, 
			tTimeout:= T#4S, 
			bBusy=> , 
			bError=> bError, 
			nErrId=> nErrorID );
		IF NOT fbSocketClose.bBusy THEN
			iState :=0;		
		END_IF
END_CASE

END_FUNCTION_BLOCK
